(* IEC 61131-3 sources: plc_generation_empirical_study/datasets/_archive/pre_native_plcverif_20260810/tasks/C09_M01_high_high_alarm_priority, 2 files *)

(* ---- interface.st ---- *)
FUNCTION_BLOCK C09_M01_high_high_alarm_priority
VAR_INPUT
    Value : REAL;
    HighLimit : REAL;
    HighHighLimit : REAL;
    Reset : BOOL;
END_VAR
VAR_OUTPUT
    HighAlarm : BOOL;
    HighHighAlarm : BOOL;
    Shutdown : BOOL;
END_VAR
END_FUNCTION_BLOCK

(* ---- reference.st ---- *)
FUNCTION_BLOCK C09_M01_high_high_alarm_priority
VAR_INPUT
    Value : REAL;
    HighLimit : REAL;
    HighHighLimit : REAL;
    Reset : BOOL;
END_VAR
VAR_OUTPUT
    HighAlarm : BOOL;
    HighHighAlarm : BOOL;
    Shutdown : BOOL;
END_VAR

IF Value >= HighHighLimit THEN
    HighAlarm := TRUE;
    HighHighAlarm := TRUE;
    Shutdown := TRUE;
ELSIF Value >= HighLimit THEN
    HighAlarm := TRUE;
END_IF;
IF Reset AND (Value < HighLimit) THEN
    HighAlarm := FALSE;
    HighHighAlarm := FALSE;
    Shutdown := FALSE;
END_IF;

END_FUNCTION_BLOCK
